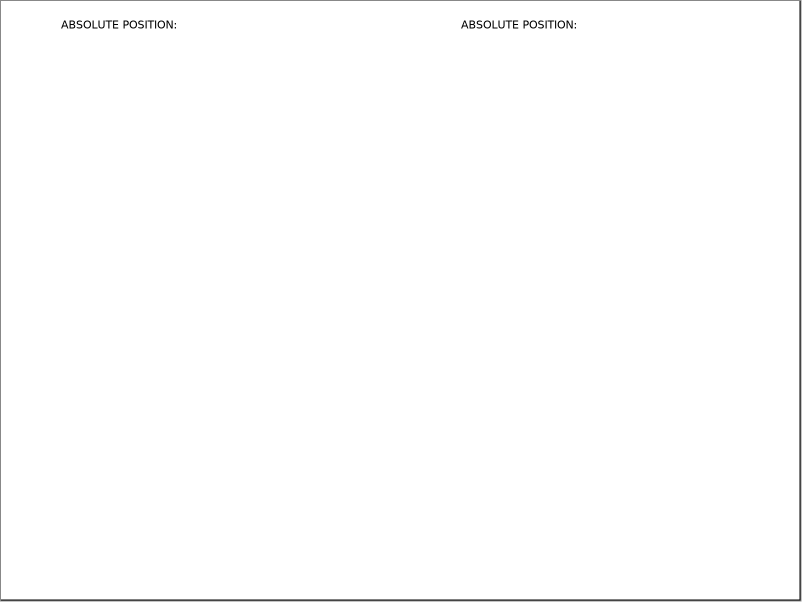
VISUALIZATION F25_Jog  // 802x602
    Rectangle (0,0 800x600)
    Label (10,10 170x30), "ABSOLUTE POSITION:"
    Label (410,10 170x30), "ABSOLUTE POSITION:"
END_VISUALIZATION

(* stored: Version 1.1.0.1, ProductVersion 3.1.4022.7
   Visu F25_Jog: Id {87b115ba-efd3-4fd4-ba68-bfbaf8f78cd7} *)
